FUNCTION_BLOCK TwoConCtlRing (* Composite Function Block Type *)
  (* Standard: 61499-2 *)
  (* Version 0.2, 2003-12-05, JHC, Rockwell Automation, Renamed from NEWCOMPFB. *)
  (* Version 0.1, 2002-01-08, JHC, Rockwell Automation, Added DLY FB as example. *)
  (* Version 0.0, 2000-05-27, JHC, Rockwell Automation *)
  (* Compiler header: package fb.rt.cs725; *)
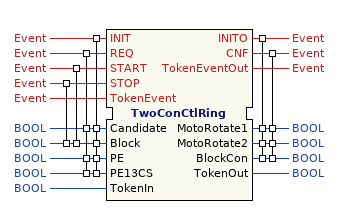
  EVENT_INPUT
    INIT WITH Candidate, Block, PE, PE13CS; (* Initialization Request *)
    REQ WITH Candidate, PE, PE13CS; (* Normal Execution Request *)
    START WITH Block;
    STOP WITH Block;
    TokenEvent;
  END_EVENT
  EVENT_OUTPUT
    INITO WITH MotoRotate1, MotoRotate2, BlockCon; (* Initialization Confirm *)
    CNF WITH MotoRotate1, MotoRotate2, BlockCon; (* Execution Confirmation *)
    TokenEventOut;
  END_EVENT
  VAR_INPUT
    Candidate : BOOL;
    Block : BOOL;
    PE : BOOL;
    PE13CS : BOOL;
    TokenIn : BOOL;
  END_VAR
  VAR_OUTPUT
    MotoRotate1 : BOOL;
    MotoRotate2 : BOOL;
    BlockCon : BOOL;
    TokenOut : BOOL;
  END_VAR
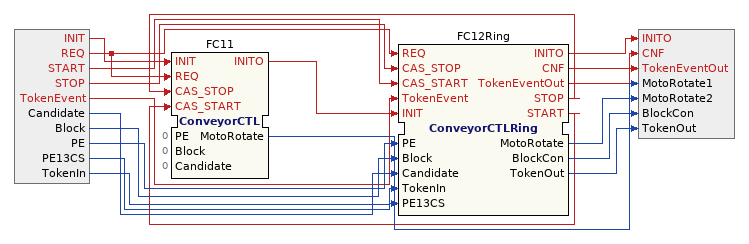
  FBS
    FC11 : ConveyorCTL(PE := 0, Block := 0, Candidate := 0);
    FC12Ring : ConveyorCTLRing;
  END_FBS
  EVENT_CONNECTIONS
    INIT TO FC11.INIT;
    REQ TO FC11.REQ;
    REQ TO FC12Ring.REQ;
    STOP TO FC12Ring.CAS_STOP;
    START TO FC12Ring.CAS_START;
    TokenEvent TO FC12Ring.TokenEvent;
    FC12Ring.INITO TO INITO;
    FC12Ring.CNF TO CNF;
    FC12Ring.TokenEventOut TO TokenEventOut;
    FC11.INITO TO FC12Ring.INIT;
    FC12Ring.STOP TO FC11.CAS_STOP;
    FC12Ring.START TO FC11.CAS_START;
  END_CONNECTIONS
  DATA_CONNECTIONS
    FC11.MotoRotate TO MotoRotate1;
    PE TO FC12Ring.PE;
    Block TO FC12Ring.Block;
    Candidate TO FC12Ring.Candidate;
    TokenIn TO FC12Ring.TokenIn;
    FC12Ring.MotoRotate TO MotoRotate2;
    FC12Ring.BlockCon TO BlockCon;
    FC12Ring.TokenOut TO TokenOut;
    PE13CS TO FC12Ring.PE13CS;
  END_CONNECTIONS
END_FUNCTION_BLOCK
